% RSLogix 500 project NW_JUICE.RSS, saved by version 12.00.00.00 %
PROJECT "3130"    % processor: MicroLogix 1400 %

PROGRAM FILES
  LAD 2   8 rungs
  LAD 3   18 rungs
  LAD 4   19 rungs
  LAD 5   13 rungs
  LAD 6   59 rungs
  LAD 8   8 rungs
  LAD 9   104 rungs
  LAD 10   28 rungs
  LAD 11, 13: only END

DATA FILES
  O0 OUTPUT  6 elements
  I1 INPUT  9 elements
  S2 STATUS  66 elements
  B3 BINARY  28 elements
  T4 TIMER  40 elements
  C5 COUNTER  5 elements
  R6 CONTROL  1 elements
  N7 INTEGER  240 elements
  F8 FLOAT  25 elements
  N9   25 elements
  N10   232 elements
  MG11   50 elements
  N12   2 elements
  N13   16 elements
  F14   21 elements
  F15   21 elements
  F16   210 elements
  N17   100 elements
  F18   15 elements
  N19   15 elements
  F20   21 elements
  F21   25 elements
  F22   25 elements
  ST23   26 elements
  N24   25 elements
  N25   20 elements
  N26   20 elements
  B27   25 elements
  N28   25 elements
  ST29   50 elements
  RI30   10 elements
  MG31   150 elements
  N32   150 elements

LADDER 2
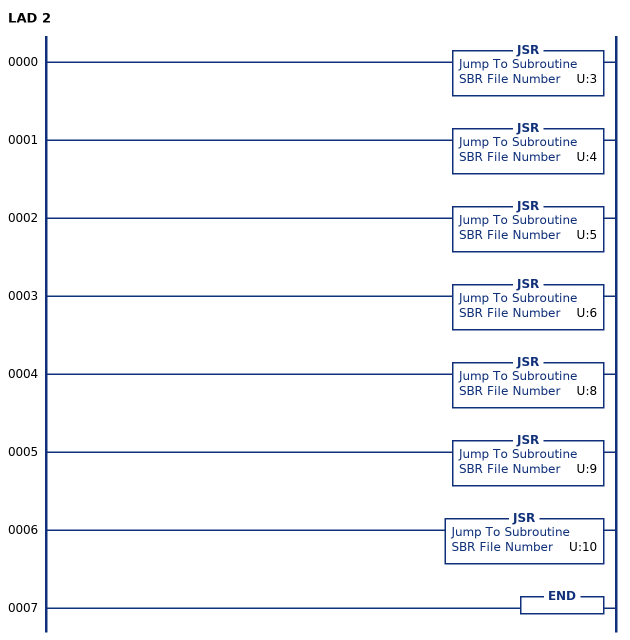
% Rung: 0 %
SOR JSR U:3 EOR
% Rung: 1 %
SOR JSR U:4 EOR
% Rung: 2 %
SOR JSR U:5 EOR
% Rung: 3 %
SOR JSR U:6 EOR
% Rung: 4 %
SOR JSR U:8 EOR
% Rung: 5 %
SOR JSR U:9 EOR
% Rung: 6 %
SOR JSR U:10 EOR
% Rung: 7 %
SOR END EOR

LADDER 3
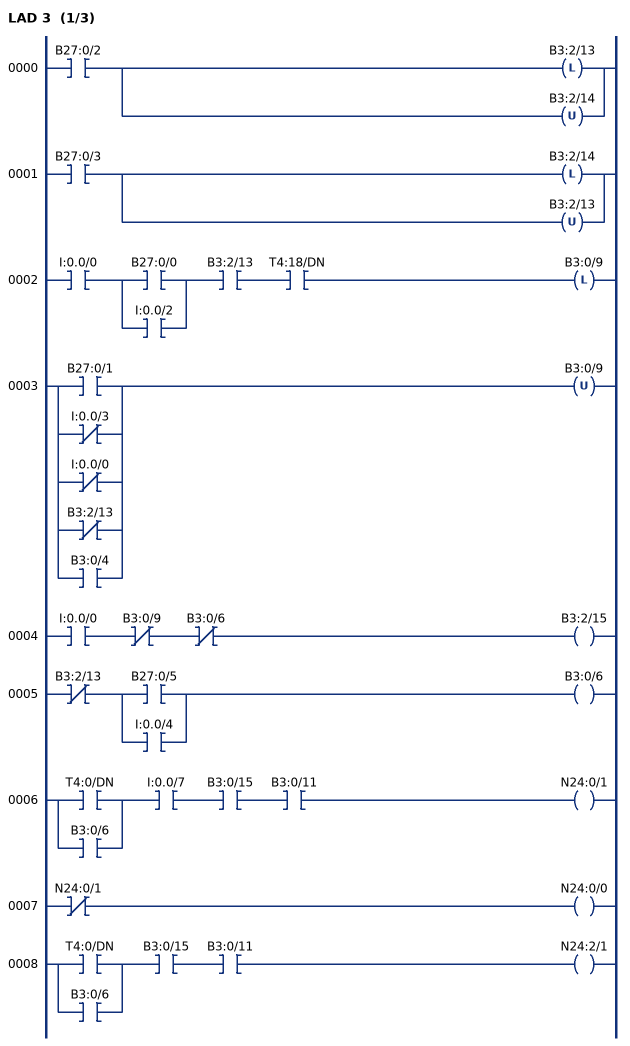
% Rung: 0 %
SOR XIC B27:0/2 BST OTL B3:2/13 NXB OTU B3:2/14 BND EOR
% Rung: 1 %
SOR XIC B27:0/3 BST OTL B3:2/14 NXB OTU B3:2/13 BND EOR
% Rung: 2 %
SOR XIC I:0.0/0 BST XIC B27:0/0 NXB XIC I:0.0/2 BND XIC B3:2/13 XIC T4:18/DN OTL B3:0/9 EOR
% Rung: 3 %
SOR BST XIC B27:0/1 NXB XIO I:0.0/3 NXB XIO I:0.0/0 NXB XIO B3:2/13 NXB XIC B3:0/4 BND OTU B3:0/9 EOR
% Rung: 4 %
SOR XIC I:0.0/0 XIO B3:0/9 XIO B3:0/6 OTE B3:2/15 EOR
% Rung: 5 %
SOR XIO B3:2/13 BST XIC B27:0/5 NXB XIC I:0.0/4 BND OTE B3:0/6 EOR
% Rung: 6 %
SOR BST XIC T4:0/DN NXB XIC B3:0/6 BND XIC I:0.0/7 XIC B3:0/15 XIC B3:0/11 OTE N24:0/1 EOR
% Rung: 7 %
SOR XIO N24:0/1 OTE N24:0/0 EOR
% Rung: 8 %
SOR BST XIC T4:0/DN NXB XIC B3:0/6 BND XIC B3:0/15 XIC B3:0/11 OTE N24:2/1 EOR

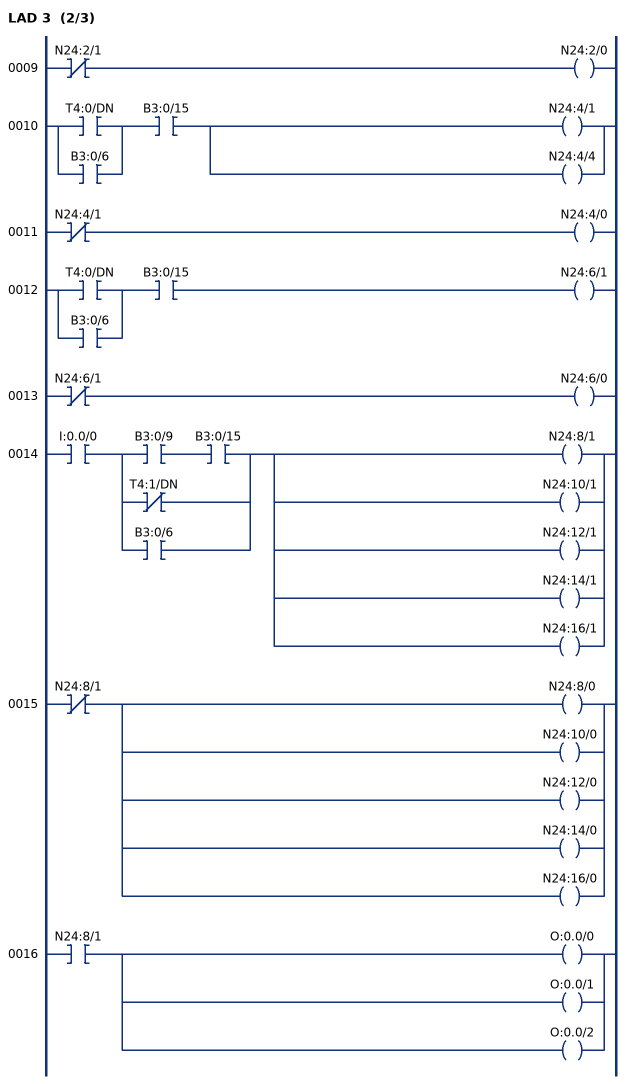
% Rung: 9 %
SOR XIO N24:2/1 OTE N24:2/0 EOR
% Rung: 10 %
SOR BST XIC T4:0/DN NXB XIC B3:0/6 BND XIC B3:0/15 BST OTE N24:4/1 NXB OTE N24:4/4 BND EOR
% Rung: 11 %
SOR XIO N24:4/1 OTE N24:4/0 EOR
% Rung: 12 %
SOR BST XIC T4:0/DN NXB XIC B3:0/6 BND XIC B3:0/15 OTE N24:6/1 EOR
% Rung: 13 %
SOR XIO N24:6/1 OTE N24:6/0 EOR
% Rung: 14 %
SOR XIC I:0.0/0 BST XIC B3:0/9 XIC B3:0/15 NXB XIO T4:1/DN NXB XIC B3:0/6 BND BST OTE N24:8/1 NXB OTE N24:10/1 NXB OTE N24:12/1 NXB OTE N24:14/1 NXB OTE N24:16/1 BND EOR
% Rung: 15 %
SOR XIO N24:8/1 BST OTE N24:8/0 NXB OTE N24:10/0 NXB OTE N24:12/0 NXB OTE N24:14/0 NXB OTE N24:16/0 BND EOR
% Rung: 16 %
SOR XIC N24:8/1 BST OTE O:0.0/0 NXB OTE O:0.0/1 NXB OTE O:0.0/2 BND EOR

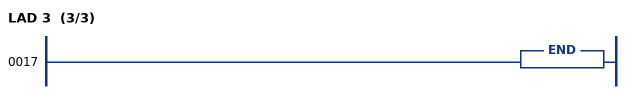
% Rung: 17 %
SOR END EOR

LADDER 4
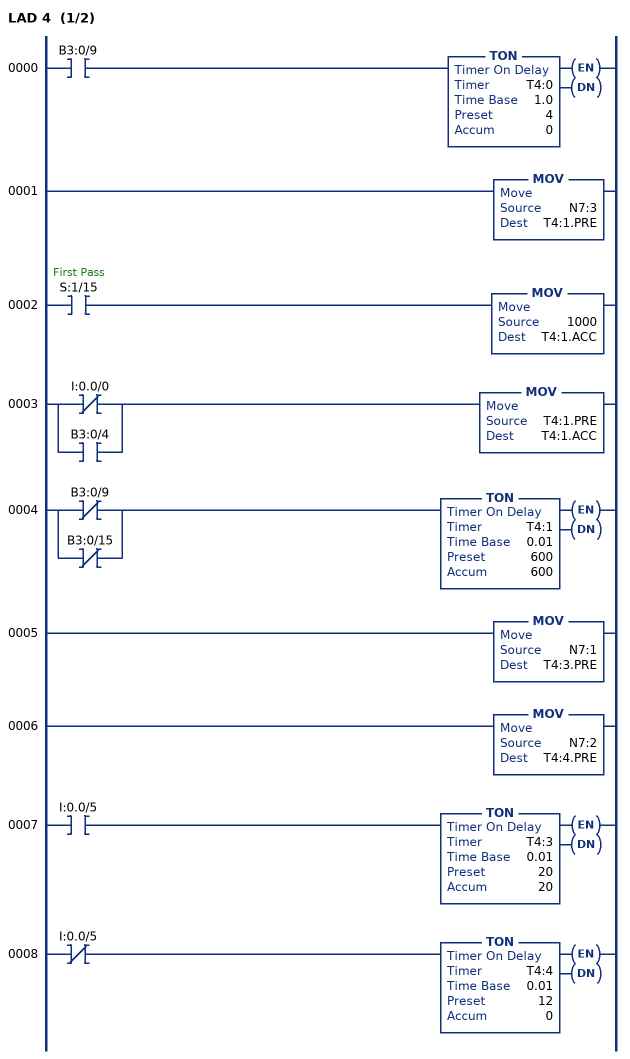
% Rung: 0 %
SOR XIC B3:0/9 TON T4:0 1.0 4 0 EOR
% Rung: 1 %
SOR MOV N7:3 T4:1.PRE EOR
% Rung: 2 %
SOR XIC S:1/15 MOV 1000 T4:1.ACC EOR
%   S:1/15  "First Pass" %
% Rung: 3 %
SOR BST XIO I:0.0/0 NXB XIC B3:0/4 BND MOV T4:1.PRE T4:1.ACC EOR
% Rung: 4 %
SOR BST XIO B3:0/9 NXB XIO B3:0/15 BND TON T4:1 0.01 600 600 EOR
% Rung: 5 %
SOR MOV N7:1 T4:3.PRE EOR
% Rung: 6 %
SOR MOV N7:2 T4:4.PRE EOR
% Rung: 7 %
SOR XIC I:0.0/5 TON T4:3 0.01 20 20 EOR
% Rung: 8 %
SOR XIO I:0.0/5 TON T4:4 0.01 12 0 EOR

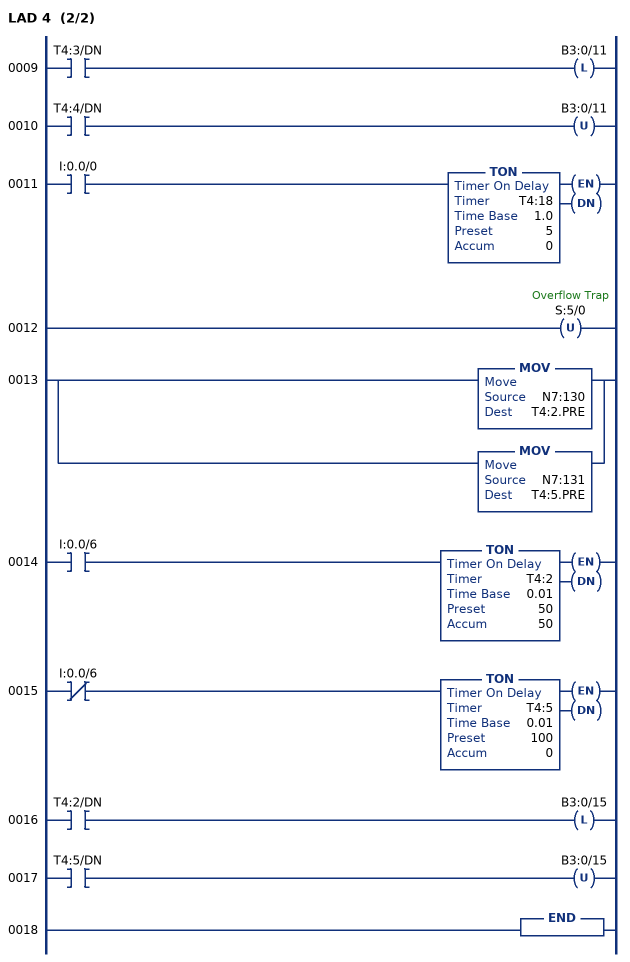
% Rung: 9 %
SOR XIC T4:3/DN OTL B3:0/11 EOR
% Rung: 10 %
SOR XIC T4:4/DN OTU B3:0/11 EOR
% Rung: 11 %
SOR XIC I:0.0/0 TON T4:18 1.0 5 0 EOR
% Rung: 12 %
SOR OTU S:5/0 EOR
%   S:5/0  "Overflow Trap" %
% Rung: 13 %
SOR BST MOV N7:130 T4:2.PRE NXB MOV N7:131 T4:5.PRE BND EOR
% Rung: 14 %
SOR XIC I:0.0/6 TON T4:2 0.01 50 50 EOR
% Rung: 15 %
SOR XIO I:0.0/6 TON T4:5 0.01 100 0 EOR
% Rung: 16 %
SOR XIC T4:2/DN OTL B3:0/15 EOR
% Rung: 17 %
SOR XIC T4:5/DN OTU B3:0/15 EOR
% Rung: 18 %
SOR END EOR

LADDER 5
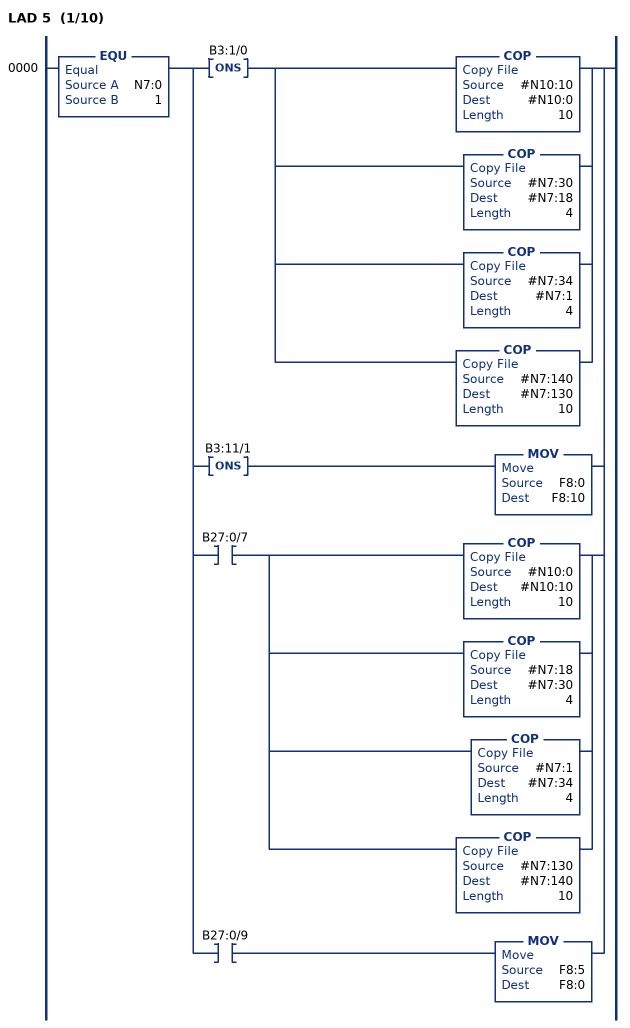
% Rung: 0 %
SOR EQU N7:0 1 BST ONS B3:1/0 BST COP #N10:10 #N10:0 10 NXB COP #N7:30 #N7:18 4 NXB COP #N7:34 #N7:1 4 NXB COP #N7:140 #N7:130 10 BND NXB ONS B3:11/1 MOV F8:0 F8:10 NXB XIC B27:0/7 BST COP #N10:0 #N10:10 10 NXB COP #N7:18 #N7:30 4 NXB COP #N7:1 #N7:34 4 NXB COP #N7:130 #N7:140 10 BND NXB XIC B27:0/9 MOV F8:5 F8:0 BND EOR

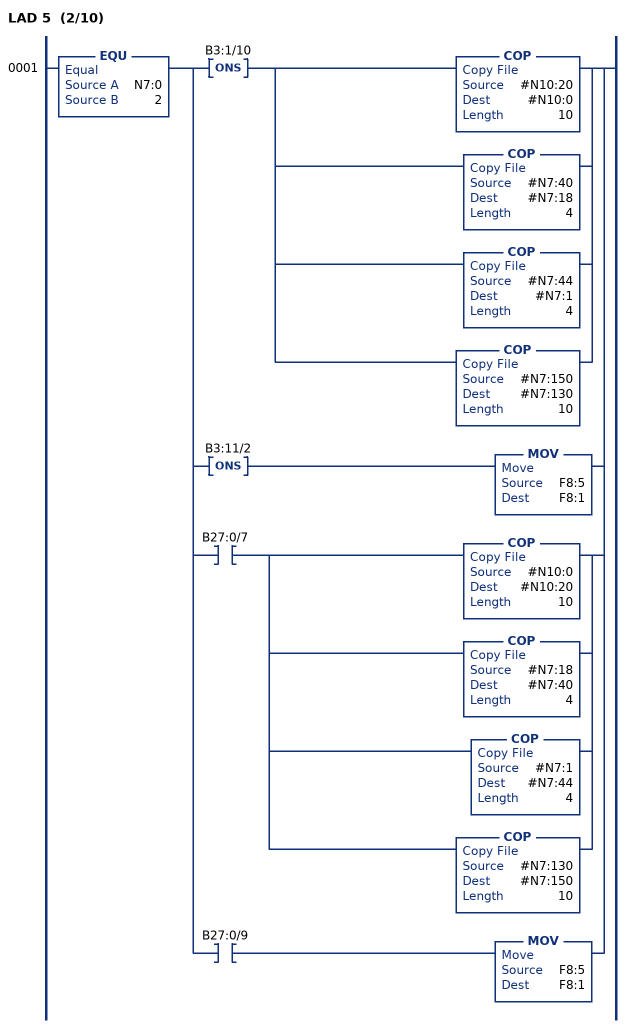
% Rung: 1 %
SOR EQU N7:0 2 BST ONS B3:1/10 BST COP #N10:20 #N10:0 10 NXB COP #N7:40 #N7:18 4 NXB COP #N7:44 #N7:1 4 NXB COP #N7:150 #N7:130 10 BND NXB ONS B3:11/2 MOV F8:5 F8:1 NXB XIC B27:0/7 BST COP #N10:0 #N10:20 10 NXB COP #N7:18 #N7:40 4 NXB COP #N7:1 #N7:44 4 NXB COP #N7:130 #N7:150 10 BND NXB XIC B27:0/9 MOV F8:5 F8:1 BND EOR

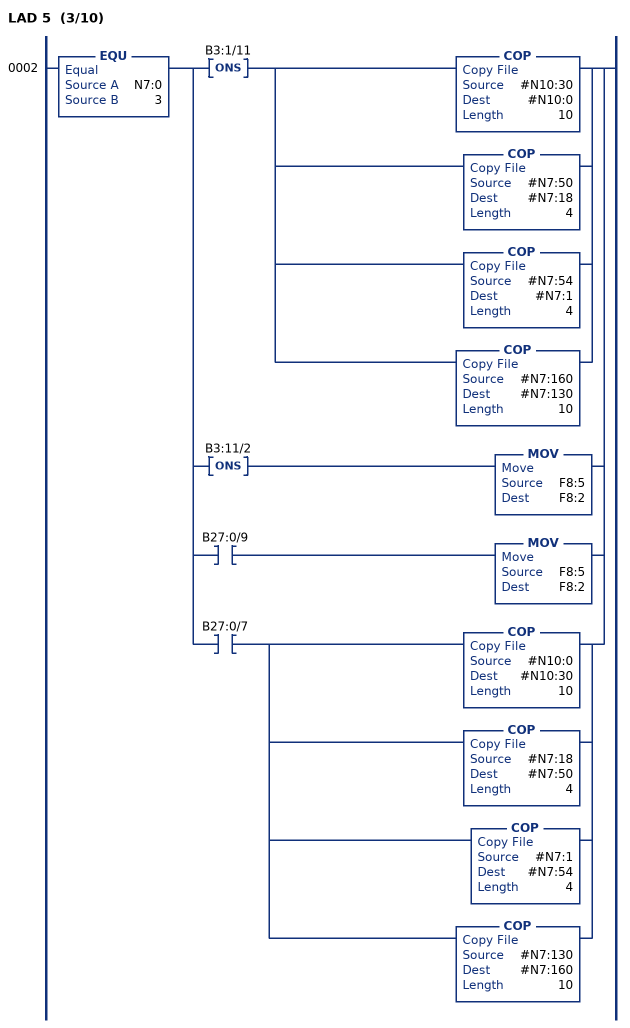
% Rung: 2 %
SOR EQU N7:0 3 BST ONS B3:1/11 BST COP #N10:30 #N10:0 10 NXB COP #N7:50 #N7:18 4 NXB COP #N7:54 #N7:1 4 NXB COP #N7:160 #N7:130 10 BND NXB ONS B3:11/2 MOV F8:5 F8:2 NXB XIC B27:0/9 MOV F8:5 F8:2 NXB XIC B27:0/7 BST COP #N10:0 #N10:30 10 NXB COP #N7:18 #N7:50 4 NXB COP #N7:1 #N7:54 4 NXB COP #N7:130 #N7:160 10 BND BND EOR

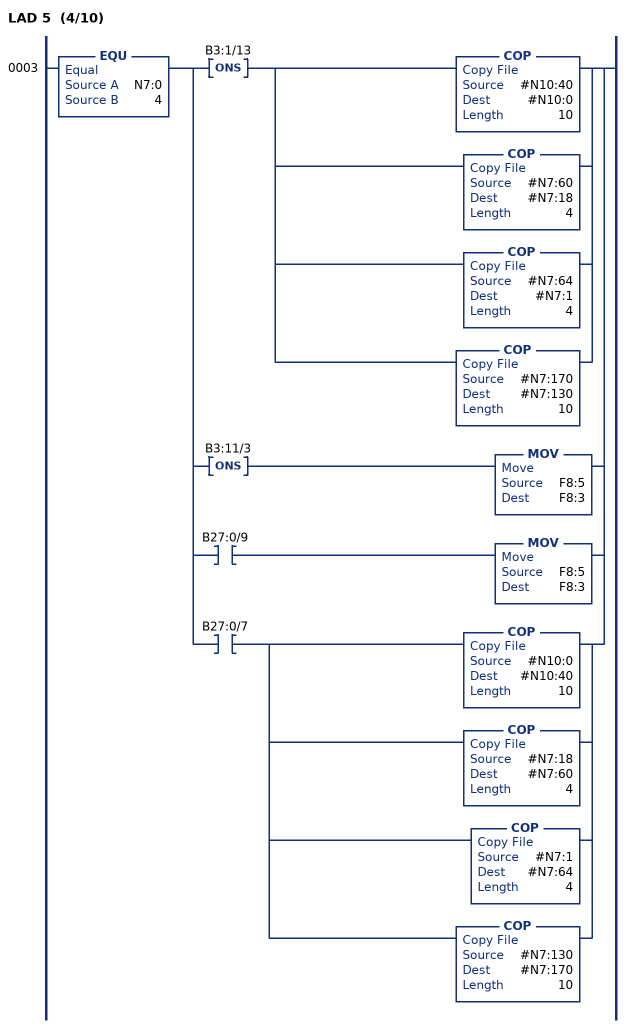
% Rung: 3 %
SOR EQU N7:0 4 BST ONS B3:1/13 BST COP #N10:40 #N10:0 10 NXB COP #N7:60 #N7:18 4 NXB COP #N7:64 #N7:1 4 NXB COP #N7:170 #N7:130 10 BND NXB ONS B3:11/3 MOV F8:5 F8:3 NXB XIC B27:0/9 MOV F8:5 F8:3 NXB XIC B27:0/7 BST COP #N10:0 #N10:40 10 NXB COP #N7:18 #N7:60 4 NXB COP #N7:1 #N7:64 4 NXB COP #N7:130 #N7:170 10 BND BND EOR

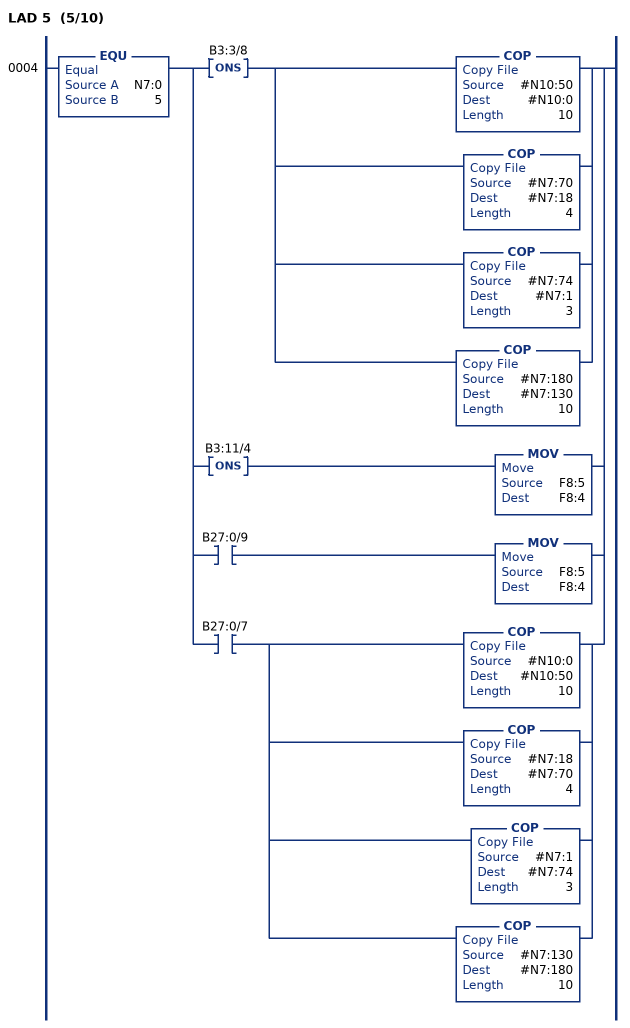
% Rung: 4 %
SOR EQU N7:0 5 BST ONS B3:3/8 BST COP #N10:50 #N10:0 10 NXB COP #N7:70 #N7:18 4 NXB COP #N7:74 #N7:1 3 NXB COP #N7:180 #N7:130 10 BND NXB ONS B3:11/4 MOV F8:5 F8:4 NXB XIC B27:0/9 MOV F8:5 F8:4 NXB XIC B27:0/7 BST COP #N10:0 #N10:50 10 NXB COP #N7:18 #N7:70 4 NXB COP #N7:1 #N7:74 3 NXB COP #N7:130 #N7:180 10 BND BND EOR

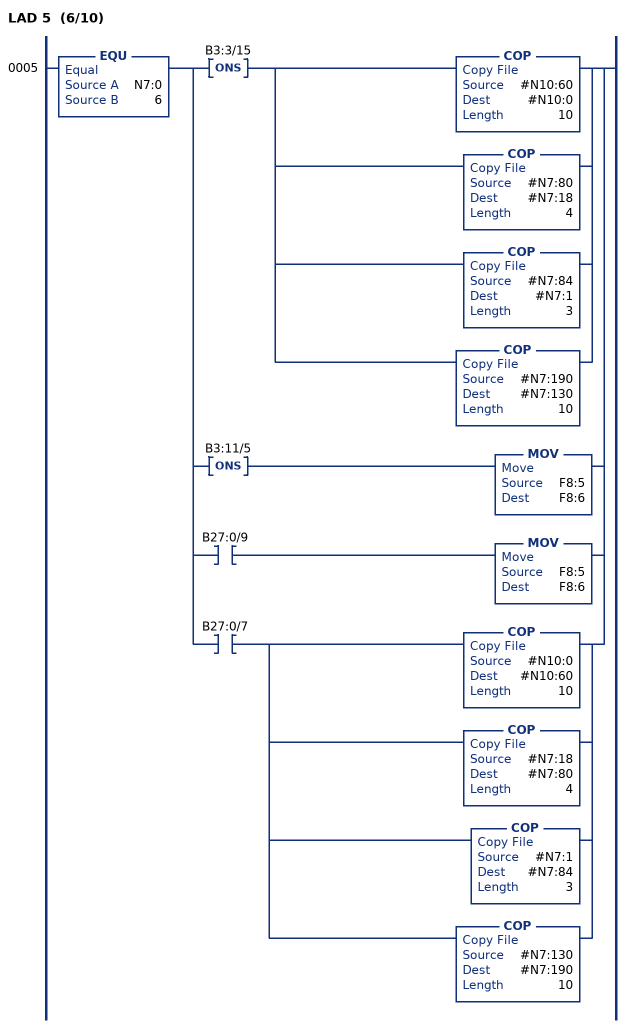
% Rung: 5 %
SOR EQU N7:0 6 BST ONS B3:3/15 BST COP #N10:60 #N10:0 10 NXB COP #N7:80 #N7:18 4 NXB COP #N7:84 #N7:1 3 NXB COP #N7:190 #N7:130 10 BND NXB ONS B3:11/5 MOV F8:5 F8:6 NXB XIC B27:0/9 MOV F8:5 F8:6 NXB XIC B27:0/7 BST COP #N10:0 #N10:60 10 NXB COP #N7:18 #N7:80 4 NXB COP #N7:1 #N7:84 3 NXB COP #N7:130 #N7:190 10 BND BND EOR

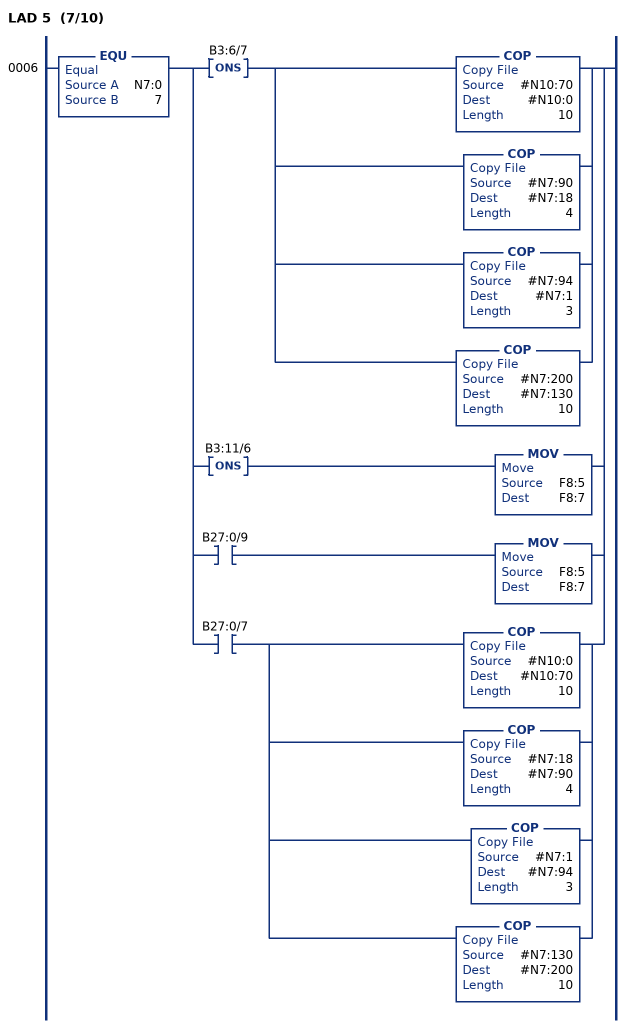
% Rung: 6 %
SOR EQU N7:0 7 BST ONS B3:6/7 BST COP #N10:70 #N10:0 10 NXB COP #N7:90 #N7:18 4 NXB COP #N7:94 #N7:1 3 NXB COP #N7:200 #N7:130 10 BND NXB ONS B3:11/6 MOV F8:5 F8:7 NXB XIC B27:0/9 MOV F8:5 F8:7 NXB XIC B27:0/7 BST COP #N10:0 #N10:70 10 NXB COP #N7:18 #N7:90 4 NXB COP #N7:1 #N7:94 3 NXB COP #N7:130 #N7:200 10 BND BND EOR

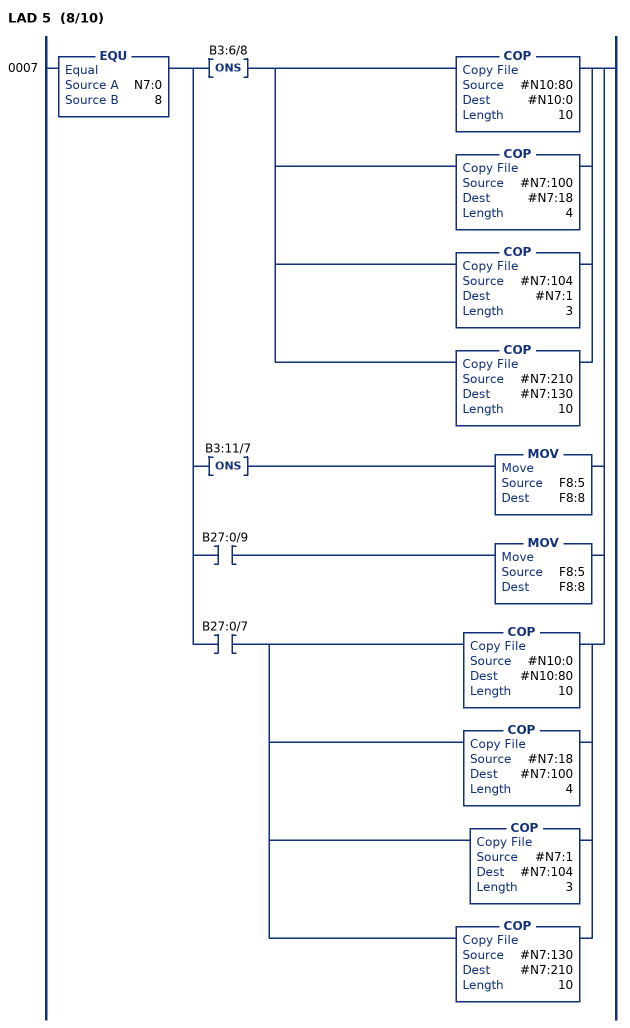
% Rung: 7 %
SOR EQU N7:0 8 BST ONS B3:6/8 BST COP #N10:80 #N10:0 10 NXB COP #N7:100 #N7:18 4 NXB COP #N7:104 #N7:1 3 NXB COP #N7:210 #N7:130 10 BND NXB ONS B3:11/7 MOV F8:5 F8:8 NXB XIC B27:0/9 MOV F8:5 F8:8 NXB XIC B27:0/7 BST COP #N10:0 #N10:80 10 NXB COP #N7:18 #N7:100 4 NXB COP #N7:1 #N7:104 3 NXB COP #N7:130 #N7:210 10 BND BND EOR

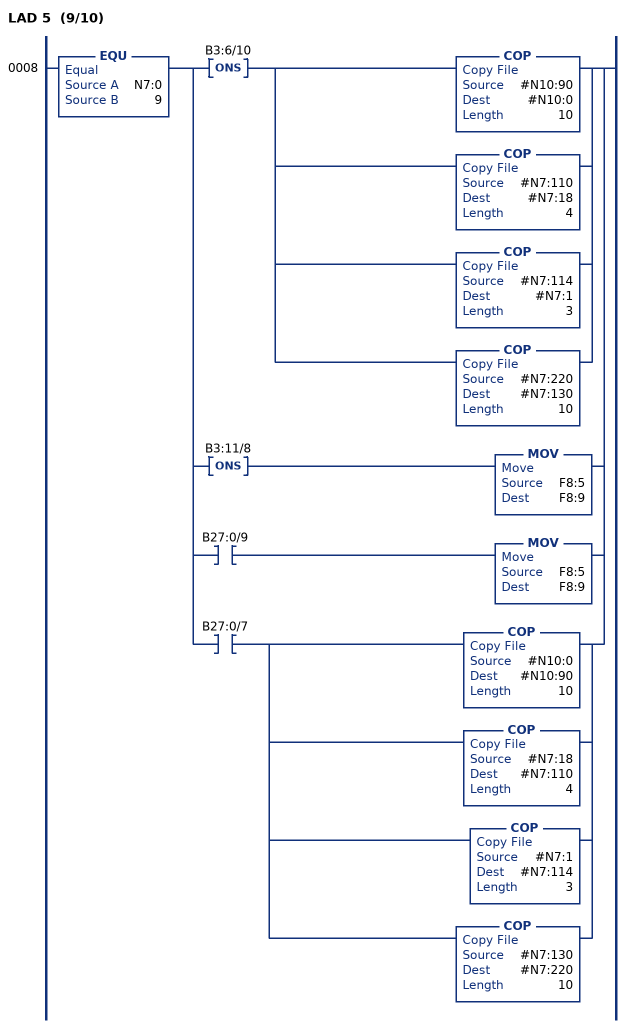
% Rung: 8 %
SOR EQU N7:0 9 BST ONS B3:6/10 BST COP #N10:90 #N10:0 10 NXB COP #N7:110 #N7:18 4 NXB COP #N7:114 #N7:1 3 NXB COP #N7:220 #N7:130 10 BND NXB ONS B3:11/8 MOV F8:5 F8:9 NXB XIC B27:0/9 MOV F8:5 F8:9 NXB XIC B27:0/7 BST COP #N10:0 #N10:90 10 NXB COP #N7:18 #N7:110 4 NXB COP #N7:1 #N7:114 3 NXB COP #N7:130 #N7:220 10 BND BND EOR

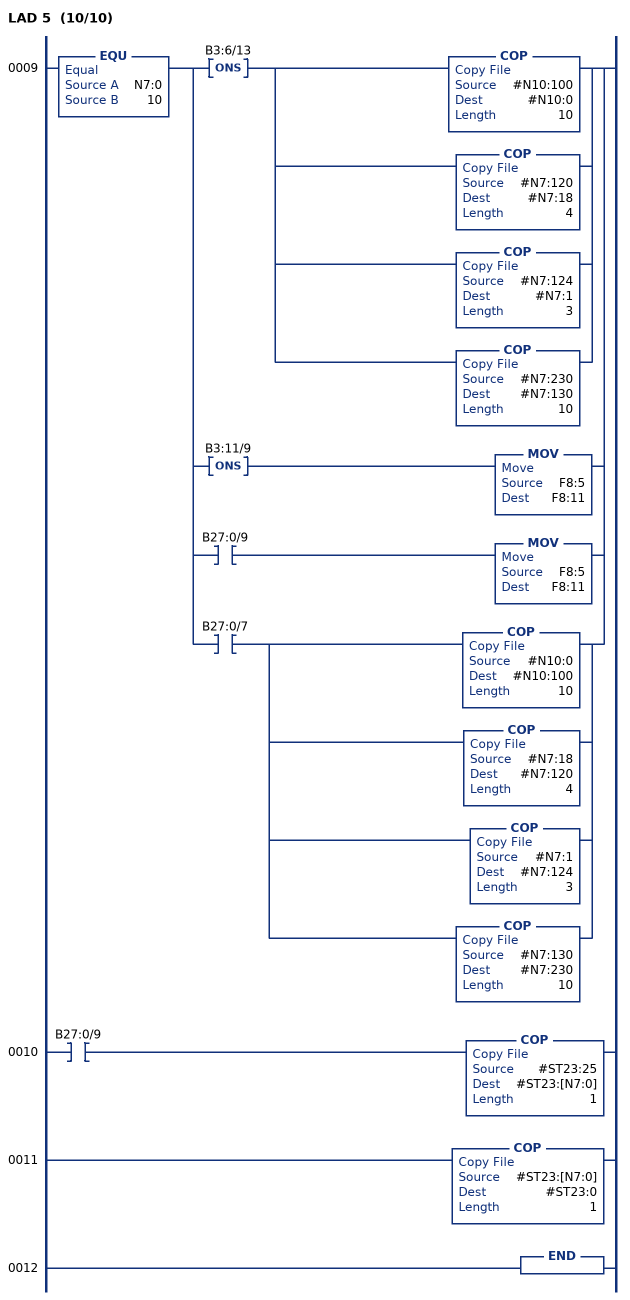
% Rung: 9 %
SOR EQU N7:0 10 BST ONS B3:6/13 BST COP #N10:100 #N10:0 10 NXB COP #N7:120 #N7:18 4 NXB COP #N7:124 #N7:1 3 NXB COP #N7:230 #N7:130 10 BND NXB ONS B3:11/9 MOV F8:5 F8:11 NXB XIC B27:0/9 MOV F8:5 F8:11 NXB XIC B27:0/7 BST COP #N10:0 #N10:100 10 NXB COP #N7:18 #N7:120 4 NXB COP #N7:1 #N7:124 3 NXB COP #N7:130 #N7:230 10 BND BND EOR
% Rung: 10 %
SOR XIC B27:0/9 COP #ST23:25 #ST23:[N7:0] 1 EOR
% Rung: 11 %
SOR COP #ST23:[N7:0] #ST23:0 1 EOR
% Rung: 12 %
SOR END EOR

LADDER 6
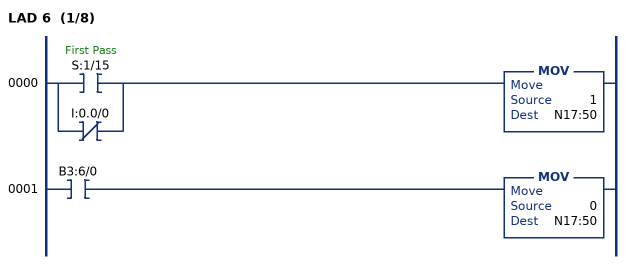
% Rung: 0 %
SOR BST XIC S:1/15 NXB XIO I:0.0/0 BND MOV 1 N17:50 EOR
%   S:1/15  "First Pass" %
% Rung: 1 %
SOR XIC B3:6/0 MOV 0 N17:50 EOR

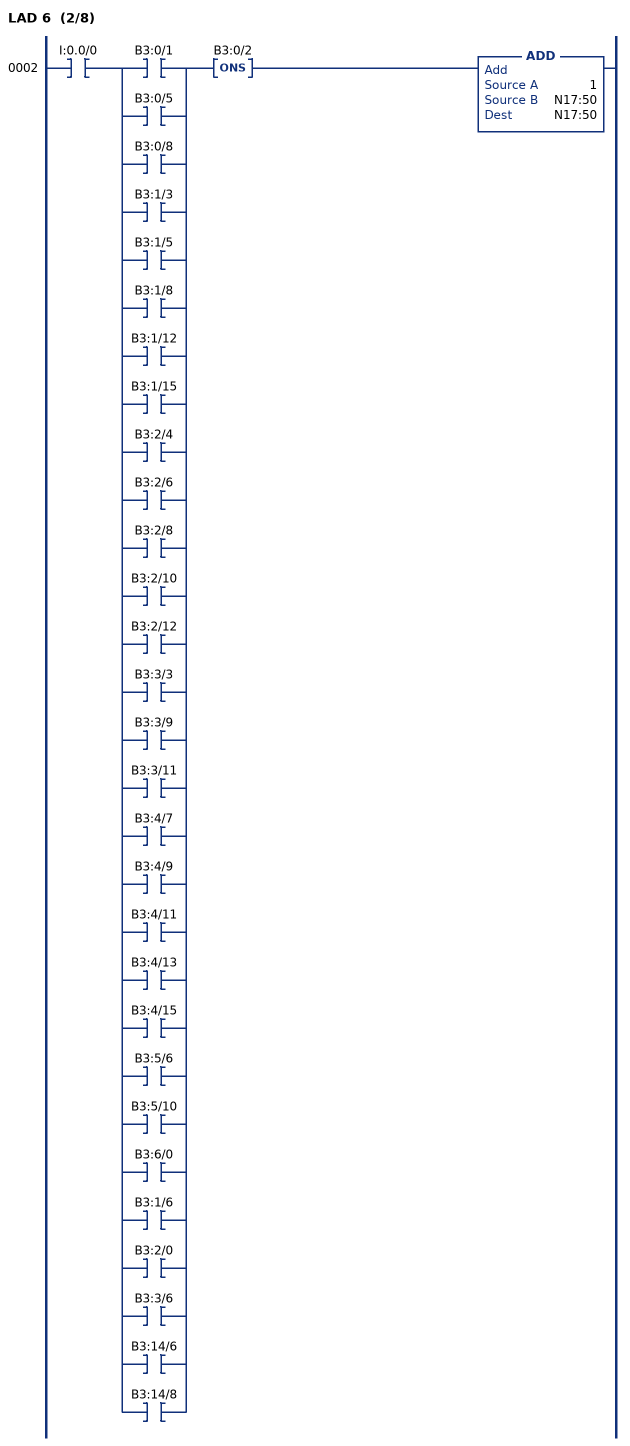
% Rung: 2 %
SOR XIC I:0.0/0 BST XIC B3:0/1 NXB XIC B3:0/5 NXB XIC B3:0/8 NXB XIC B3:1/3 NXB XIC B3:1/5 NXB XIC B3:1/8 NXB XIC B3:1/12 NXB XIC B3:1/15 NXB XIC B3:2/4 NXB XIC B3:2/6 NXB XIC B3:2/8 NXB XIC B3:2/10 NXB XIC B3:2/12 NXB XIC B3:3/3 NXB XIC B3:3/9 NXB XIC B3:3/11 NXB XIC B3:4/7 NXB XIC B3:4/9 NXB XIC B3:4/11 NXB XIC B3:4/13 NXB XIC B3:4/15 NXB XIC B3:5/6 NXB XIC B3:5/10 NXB XIC B3:6/0 NXB XIC B3:1/6 NXB XIC B3:2/0 NXB XIC B3:3/6 NXB XIC B3:14/6 NXB XIC B3:14/8 BND ONS B3:0/2 ADD 1 N17:50 N17:50 EOR

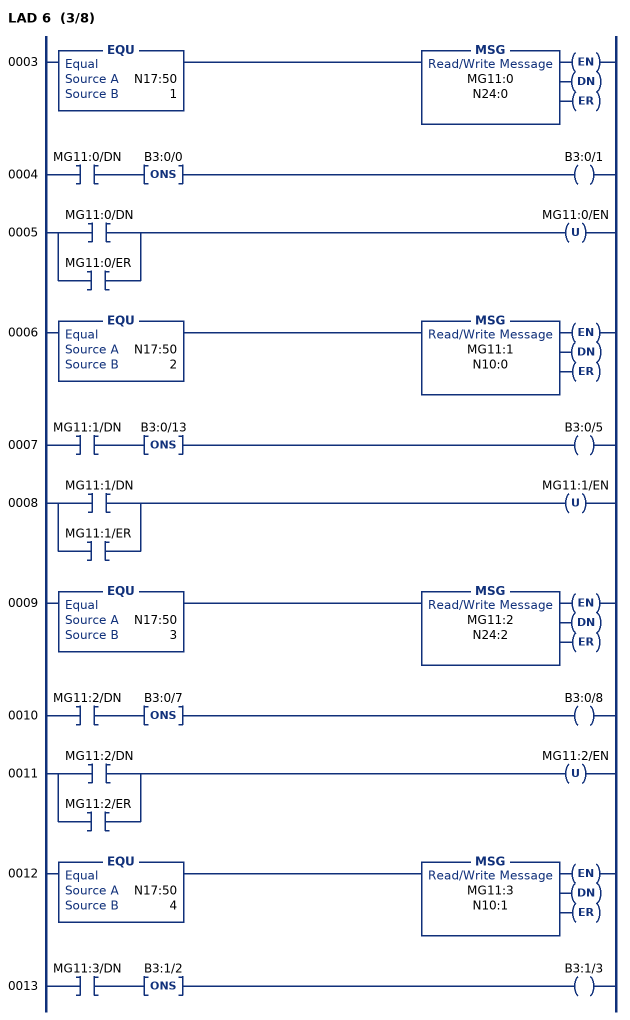
% Rung: 3 %
SOR EQU N17:50 1 MSG MG11:0 N24:0 EOR
%   MSG set-up: 06 Write Single Register (4xxxxx) | 2 | 1 | 8193 | N24:0 | 0 | 1 | 0 | CLIENT              :502 | 0 | 0 | ? %
% Rung: 4 %
SOR XIC MG11:0/DN ONS B3:0/0 OTE B3:0/1 EOR
% Rung: 5 %
SOR BST XIC MG11:0/DN NXB XIC MG11:0/ER BND OTU MG11:0/EN EOR
% Rung: 6 %
SOR EQU N17:50 2 MSG MG11:1 N10:0 EOR
%   MSG set-up: 06 Write Single Register (4xxxxx) | 2 | 1 | 8194 | N10:0 | 0 | 1 | 0 | CLIENT              :502 | 0 | 0 | ? %
% Rung: 7 %
SOR XIC MG11:1/DN ONS B3:0/13 OTE B3:0/5 EOR
% Rung: 8 %
SOR BST XIC MG11:1/DN NXB XIC MG11:1/ER BND OTU MG11:1/EN EOR
% Rung: 9 %
SOR EQU N17:50 3 MSG MG11:2 N24:2 EOR
%   MSG set-up: 06 Write Single Register (4xxxxx) | 2 | 1 | 8193 | N24:2 | 0 | 2 | 0 | CLIENT              :502 | 0 | 0 | ? %
% Rung: 10 %
SOR XIC MG11:2/DN ONS B3:0/7 OTE B3:0/8 EOR
% Rung: 11 %
SOR BST XIC MG11:2/DN NXB XIC MG11:2/ER BND OTU MG11:2/EN EOR
% Rung: 12 %
SOR EQU N17:50 4 MSG MG11:3 N10:1 EOR
%   MSG set-up: 06 Write Single Register (4xxxxx) | 2 | 1 | 8194 | N10:1 | 0 | 2 | 0 | CLIENT              :502 | 0 | 0 | ? %
% Rung: 13 %
SOR XIC MG11:3/DN ONS B3:1/2 OTE B3:1/3 EOR

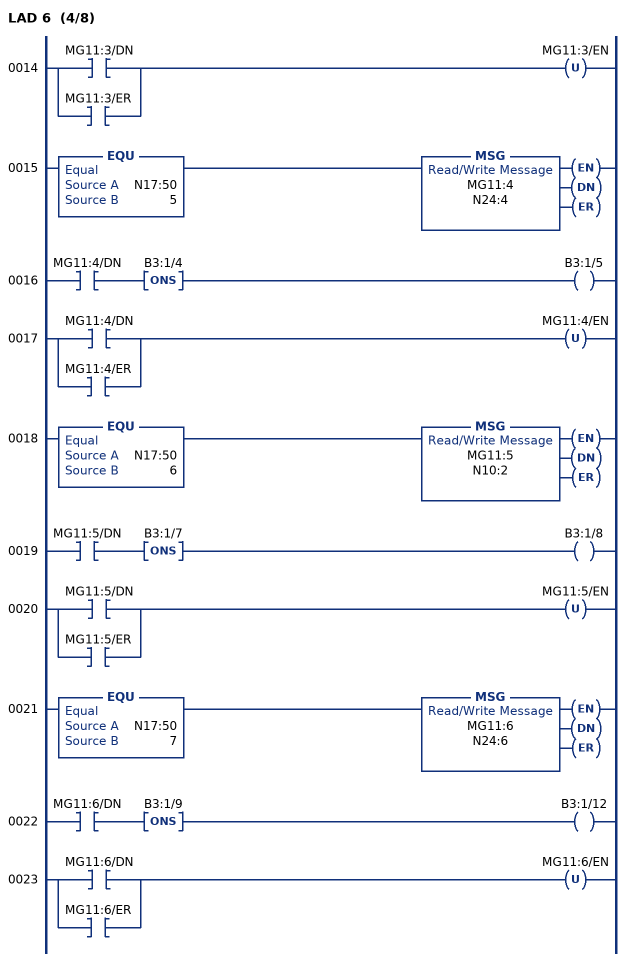
% Rung: 14 %
SOR BST XIC MG11:3/DN NXB XIC MG11:3/ER BND OTU MG11:3/EN EOR
% Rung: 15 %
SOR EQU N17:50 5 MSG MG11:4 N24:4 EOR
%   MSG set-up: 06 Write Single Register (4xxxxx) | 2 | 1 | 8193 | N24:4 | 0 | 3 | 0 | CLIENT              :502 | 0 | 0 | ? %
% Rung: 16 %
SOR XIC MG11:4/DN ONS B3:1/4 OTE B3:1/5 EOR
% Rung: 17 %
SOR BST XIC MG11:4/DN NXB XIC MG11:4/ER BND OTU MG11:4/EN EOR
% Rung: 18 %
SOR EQU N17:50 6 MSG MG11:5 N10:2 EOR
%   MSG set-up: 06 Write Single Register (4xxxxx) | 2 | 1 | 8194 | N10:2 | 0 | 3 | 0 | CLIENT              :502 | 0 | 0 | ? %
% Rung: 19 %
SOR XIC MG11:5/DN ONS B3:1/7 OTE B3:1/8 EOR
% Rung: 20 %
SOR BST XIC MG11:5/DN NXB XIC MG11:5/ER BND OTU MG11:5/EN EOR
% Rung: 21 %
SOR EQU N17:50 7 MSG MG11:6 N24:6 EOR
%   MSG set-up: 06 Write Single Register (4xxxxx) | 2 | 1 | 8193 | N24:6 | 0 | 4 | 0 | CLIENT              :502 | 0 | 0 | ? %
% Rung: 22 %
SOR XIC MG11:6/DN ONS B3:1/9 OTE B3:1/12 EOR
% Rung: 23 %
SOR BST XIC MG11:6/DN NXB XIC MG11:6/ER BND OTU MG11:6/EN EOR

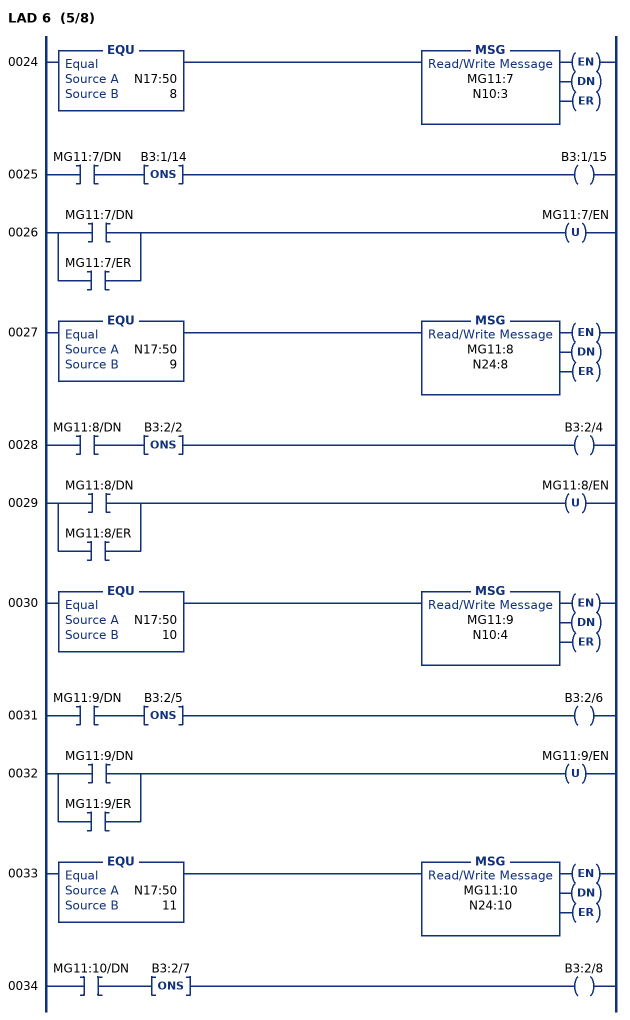
% Rung: 24 %
SOR EQU N17:50 8 MSG MG11:7 N10:3 EOR
%   MSG set-up: 06 Write Single Register (4xxxxx) | 2 | 1 | 8194 | N10:3 | 0 | 4 | 0 | CLIENT              :502 | 0 | 0 | ? %
% Rung: 25 %
SOR XIC MG11:7/DN ONS B3:1/14 OTE B3:1/15 EOR
% Rung: 26 %
SOR BST XIC MG11:7/DN NXB XIC MG11:7/ER BND OTU MG11:7/EN EOR
% Rung: 27 %
SOR EQU N17:50 9 MSG MG11:8 N24:8 EOR
%   MSG set-up: 06 Write Single Register (4xxxxx) | 2 | 1 | 8193 | N24:8 | 0 | 5 | 0 | CLIENT              :502 | 0 | 0 | ? %
% Rung: 28 %
SOR XIC MG11:8/DN ONS B3:2/2 OTE B3:2/4 EOR
% Rung: 29 %
SOR BST XIC MG11:8/DN NXB XIC MG11:8/ER BND OTU MG11:8/EN EOR
% Rung: 30 %
SOR EQU N17:50 10 MSG MG11:9 N10:4 EOR
%   MSG set-up: 06 Write Single Register (4xxxxx) | 2 | 1 | 8194 | N10:4 | 0 | 5 | 0 | CLIENT              :502 | 0 | 0 | ? %
% Rung: 31 %
SOR XIC MG11:9/DN ONS B3:2/5 OTE B3:2/6 EOR
% Rung: 32 %
SOR BST XIC MG11:9/DN NXB XIC MG11:9/ER BND OTU MG11:9/EN EOR
% Rung: 33 %
SOR EQU N17:50 11 MSG MG11:10 N24:10 EOR
%   MSG set-up: 06 Write Single Register (4xxxxx) | 2 | 1 | 8193 | N24:10 | 0 | 6 | 0 | CLIENT              :502 | 0 | 0 | ? %
% Rung: 34 %
SOR XIC MG11:10/DN ONS B3:2/7 OTE B3:2/8 EOR

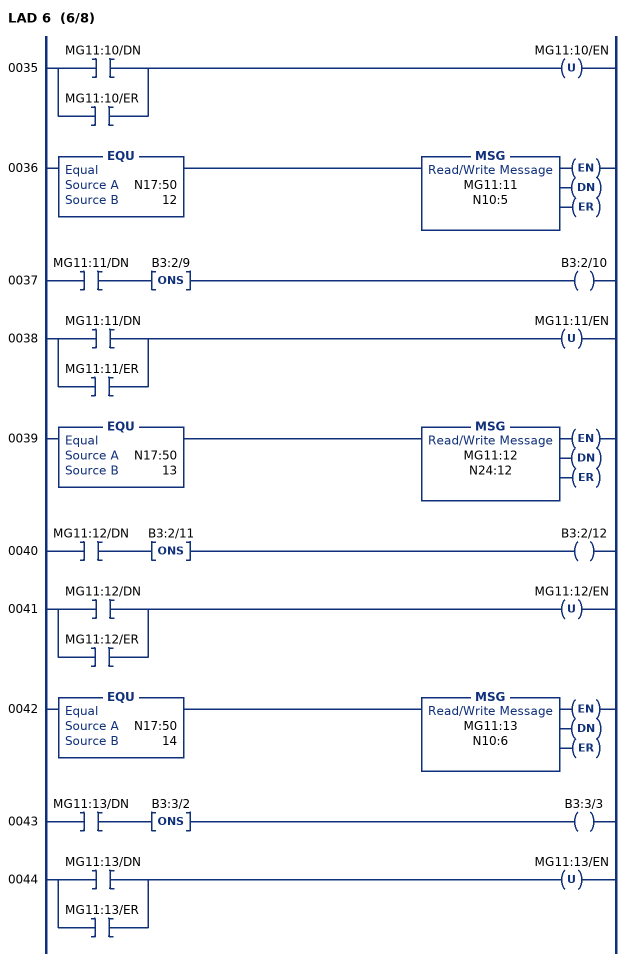
% Rung: 35 %
SOR BST XIC MG11:10/DN NXB XIC MG11:10/ER BND OTU MG11:10/EN EOR
% Rung: 36 %
SOR EQU N17:50 12 MSG MG11:11 N10:5 EOR
%   MSG set-up: 06 Write Single Register (4xxxxx) | 2 | 1 | 8194 | N10:5 | 0 | 6 | 0 | CLIENT              :502 | 0 | 0 | ? %
% Rung: 37 %
SOR XIC MG11:11/DN ONS B3:2/9 OTE B3:2/10 EOR
% Rung: 38 %
SOR BST XIC MG11:11/DN NXB XIC MG11:11/ER BND OTU MG11:11/EN EOR
% Rung: 39 %
SOR EQU N17:50 13 MSG MG11:12 N24:12 EOR
%   MSG set-up: 06 Write Single Register (4xxxxx) | 2 | 1 | 8193 | N24:12 | 0 | 7 | 0 | CLIENT              :502 | 0 | 0 | ? %
% Rung: 40 %
SOR XIC MG11:12/DN ONS B3:2/11 OTE B3:2/12 EOR
% Rung: 41 %
SOR BST XIC MG11:12/DN NXB XIC MG11:12/ER BND OTU MG11:12/EN EOR
% Rung: 42 %
SOR EQU N17:50 14 MSG MG11:13 N10:6 EOR
%   MSG set-up: 06 Write Single Register (4xxxxx) | 2 | 1 | 8194 | N10:6 | 0 | 7 | 0 | CLIENT              :502 | 0 | 0 | ? %
% Rung: 43 %
SOR XIC MG11:13/DN ONS B3:3/2 OTE B3:3/3 EOR
% Rung: 44 %
SOR BST XIC MG11:13/DN NXB XIC MG11:13/ER BND OTU MG11:13/EN EOR

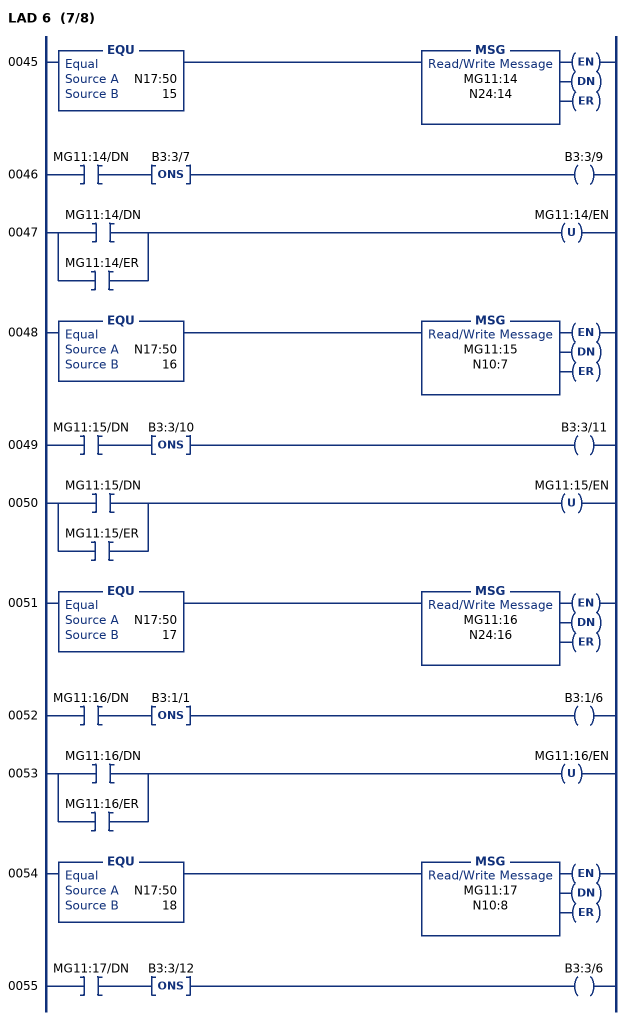
% Rung: 45 %
SOR EQU N17:50 15 MSG MG11:14 N24:14 EOR
%   MSG set-up: 06 Write Single Register (4xxxxx) | 2 | 1 | 8193 | N24:14 | 0 | 8 | 0 | CLIENT              :502 | 0 | 0 | ? %
% Rung: 46 %
SOR XIC MG11:14/DN ONS B3:3/7 OTE B3:3/9 EOR
% Rung: 47 %
SOR BST XIC MG11:14/DN NXB XIC MG11:14/ER BND OTU MG11:14/EN EOR
% Rung: 48 %
SOR EQU N17:50 16 MSG MG11:15 N10:7 EOR
%   MSG set-up: 06 Write Single Register (4xxxxx) | 2 | 1 | 8194 | N10:7 | 0 | 8 | 0 | CLIENT              :502 | 0 | 0 | ? %
% Rung: 49 %
SOR XIC MG11:15/DN ONS B3:3/10 OTE B3:3/11 EOR
% Rung: 50 %
SOR BST XIC MG11:15/DN NXB XIC MG11:15/ER BND OTU MG11:15/EN EOR
% Rung: 51 %
SOR EQU N17:50 17 MSG MG11:16 N24:16 EOR
%   MSG set-up: 06 Write Single Register (4xxxxx) | 2 | 1 | 8193 | N24:16 | 0 | 9 | 0 | CLIENT              :502 | 0 | 0 | ? %
% Rung: 52 %
SOR XIC MG11:16/DN ONS B3:1/1 OTE B3:1/6 EOR
% Rung: 53 %
SOR BST XIC MG11:16/DN NXB XIC MG11:16/ER BND OTU MG11:16/EN EOR
% Rung: 54 %
SOR EQU N17:50 18 MSG MG11:17 N10:8 EOR
%   MSG set-up: 06 Write Single Register (4xxxxx) | 2 | 1 | 8194 | N10:8 | 0 | 9 | 0 | CLIENT              :502 | 0 | 0 | ? %
% Rung: 55 %
SOR XIC MG11:17/DN ONS B3:3/12 OTE B3:3/6 EOR

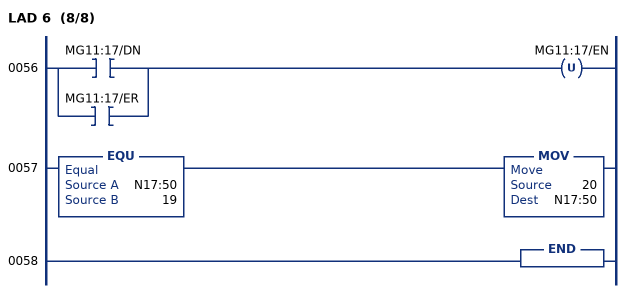
% Rung: 56 %
SOR BST XIC MG11:17/DN NXB XIC MG11:17/ER BND OTU MG11:17/EN EOR
% Rung: 57 %
SOR EQU N17:50 19 MOV 20 N17:50 EOR
% Rung: 58 %
SOR END EOR

LADDER 8
